SUBAPPLICATION Uebung_033_sub (* LED Strip Blinkende LED *)
  (* Standard: 61499-2; Description: Copyright (c) 2023 Meisterschulen am Ostbahnhof This program and the accompanying materials are made available under the terms of the Eclipse Public License 2.0 which is available at https://www.eclipse.org/legal/epl-2.0/ SPDX-License-Identifier: EPL-2.0 *)
  (* Version 1.0, 2023-10-23, Franz Höpfinger, Meisterschulen am Ostbahnhof *)
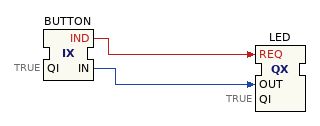
  FBS
    LED : QX(QI := TRUE);
    BUTTON : IX(QI := TRUE);
  END_FBS
  EVENT_CONNECTIONS
    BUTTON.IND TO LED.REQ;
  END_CONNECTIONS
  DATA_CONNECTIONS
    BUTTON.IN TO LED.OUT;
  END_CONNECTIONS
END_SUBAPPLICATION
